Yaskawa INFORM job: MT_OPEN-DOOR.JBI

/JOB
//NAME MT_OPEN-DOOR
//POS
///NPOS 0,0,0,0,0,0
//INST
///DATE 2023/11/28 18:35
///ATTR SC,RW
///GROUP1 RB1
NOP
DOUT OT#(530) OFF
TIMER T=0.100
DOUT OT#(530) ON
TIMER T=0.100
DOUT OT#(530) OFF
COMM WAIT IN#(530)=ON
END
